// TIA Portal V16 export
// export: Created 2024-09-05T17:39:17.7617782Z, ExportSetting WithDefaults, DisplayName Totally Integrated Automation Portal, DisplayVersion V16 Update 6, DisplayName TIA Portal Version Control Interface, DisplayVersion V16 Update 2, DisplayName TIA Portal Openness, DisplayVersion V16 Update 6, DisplayName STEP 7 Professional, DisplayVersion V16 Update 6, DisplayName STEP 7 Safety, DisplayVersion V16, DisplayName WinCC Advanced, DisplayVersion V16 Update 6
DATA_BLOCK "ParametersLimits_DB"   // DB40
VERSION : 0.1
// stored: AutoNumber true, DBAccessibleFromOPCUA true, InstanceOfName ParametersLimits, InstanceOfType FB
"ParametersLimits"
   // VAR RETAIN
   //    limits : "udt_parametersLimits";
   // END_VAR
BEGIN
   limits.ServoPositions[0].min := 5000;
   limits.ServoPositions[1].min := 780000;
   limits.ServoPositions[2].min := 1508000;
   limits.ServoPositions[3..9].min := 0;
   limits.ServoPositions[0].max := 15000;
   limits.ServoPositions[1].max := 790000;
   limits.ServoPositions[2].max := 1518000;
   limits.ServoPositions[3..9].max := 0;
END_DATA_BLOCK
